TYPE E_AutoStep :
(
    Idle              := 0,
    CheckReady        := 10,
    TrayFeed          := 20,
    PickProduct       := 30,
    TopVisionAngle    := 40,
    RotateProduct     := 50,
    PlaceToRing       := 60,
    RingToClamp       := 70,
    ClampProduct      := 80,
    CoaxVision        := 90,
    CoaxAdjust        := 100,
    ScrewMove         := 110,
    ScrewTighten      := 120,
    RingReturn        := 130,
    PickBack          := 140,
    PlaceToTray       := 150,
    NextProduct       := 160,
    Finished          := 170,
    Error             := 999
);
END_TYPE

(* stored: Version 1.1.0.1, ProductVersion 3.1.4026.18
   DUT E_AutoStep: Id {2824ac1e-3866-4ca8-8673-088a023ae5b0} *)
